FUNCTION_BLOCK T_CommandQueue_GetNextCommandNormalPriorityWithLowPriority_ReturnTrue EXTENDS T_UnitTestBase
VAR
  commandLowPriority : T_CommandTask;
  commandNormalPriority : T_CommandTask;
  commandQueue : T_CommandQueue;
  myTestState, prevState : (ARRANGE, ACT, ASSERT);
  actual : I_Task;
  expected : I_Task;
END_VAR

CASE myTestState OF
  ARRANGE:
  	expected := commandNormalPriority;
	commandQueue.Clear();
	commandQueue.AddNormalPriority(commandNormalPriority);
	commandQueue.AddLowPriority(commandLowPriority);
    myTestState := ACT;
  
  ACT:
    commandQueue.GetNext(output_command => actual);
	myTestState := ASSERT;
	
  ASSERT:
    assertion.AssertEquals_INTERFACE(expected, actual, 'commandQueue.GetNext high priority with Low priority = TRUE');
    myTestState := ARRANGE;
    TestFinished();
END_CASE

END_FUNCTION_BLOCK

(* stored: Version 1.1.0.1, ProductVersion 3.1.4024.12
   POU T_CommandQueue_GetNextCommandNormalPriorityWithLowPriority_ReturnTrue: Id {3a0b4056-83ee-45fb-b2fa-f7c0c9cf6fd2}, SpecialFunc None *)
